FUNCTION MatTimesRPS : RobotPoseSimple
VAR_INPUT
	K: ARRAY [0..2,0..2] OF LREAL;
	pose: RobotPoseSimple;
END_VAR

//2.) apply gain on errors
MatTimesRPS.x 	 := K[0,0] * pose.x + K[1,0] * pose.y + K[2,0] * pose.theta;
MatTimesRPS.y 	 := K[0,1] * pose.x + K[1,1] * pose.y + K[2,1] * pose.theta;
MatTimesRPS.theta := K[0,2] * pose.x + K[1,2] * pose.y + K[2,2] * pose.theta;

END_FUNCTION

(* stored: Version 1.1.0.1, ProductVersion 3.1.4024.11
   POU MatTimesRPS: Id {d8a25963-196a-479f-8502-ec67bf6c40a1}, SpecialFunc None *)
